PROGRAM MAIN
VAR
	tonCycle			: TON; //timer used to measure 1min period
	fbSceneController	: FB_SceneController;
	fbPBL				: FB_PBL; //previous brightness level data block
END_VAR

//init timer and set dimm value for all street lamps every 1M
//in other words: repeat control signal in case of power failure
tonCycle(IN := NOT tonCycle.Q, PT:=T#1M, Q=>GVL_StreetLamps.bSetDimmValue);

//assign DALI addresses at the begining of the program
P_AddrAssignment();

P_BACnet_Manual();
P_BACnet_ActualLevel();
P_BACnet_Error();
P_BACnet_Level();
P_BACnet_Motion();
P_BACnet_Scene();

//KNX motion sensors activated
P_MotionSensors(bEnable := TRUE);

//listen to alarm
P_AlarmMode();

//if there is no alarm
IF NOT fbBACnet_BV_Alarm.bPresentValue THEN
	//maintain auto mode and scene control
	P_AutoMode();
	fbSceneController();
END_IF

END_PROGRAM

(* stored: Version 1.1.0.1, ProductVersion 3.1.4024.5
   POU MAIN: Id {18ca1070-638d-4130-82d4-030f23fa1969}, SpecialFunc None *)
